TYPE U_INSTANCE_CTRL :
UNION
  stCtrl              : ARRAY[1..MAX_PROCESS] OF ST_INSTANCE_CTRL;
  byCtrl    AT %I*    : ARRAY[1..MAX_PROCESS] OF
                        ARRAY[1..SIZEOF(ST_INSTANCE_CTRL)] OF BYTE;
END_UNION
END_TYPE

(* stored: Version 1.1.0.1, ProductVersion 3.1.4026.13
   DUT U_INSTANCE_CTRL: Id {47c175a7-2bcc-4724-8624-6df1a10edb8b} *)
